LIN {X 0,Y 116.335,Z 316.276,A -85,B 0,C 180,E1 -30784.417,E2 -30784.417} C_VEL
LIN {X 0,Y 111.111,Z 327.603,A -85,B 0,C 180,E1 -30784.983,E2 -30784.983} C_VEL
LIN {X 0,Y 104.199,Z 339.212,A -85,B 0,C 180,E1 -30785.813,E2 -30785.813} C_VEL
LIN {X 0,Y 96.428,Z 349.65,A -85,B 0,C 180,E1 -30786.768,E2 -30786.768} C_VEL
LIN {X 0,Y 88.698,Z 358.177,A -85,B 0,C 180,E1 -30787.928,E2 -30787.928} C_VEL
LIN {X 0,Y 80.178,Z 366.031,A -85,B 0,C 180,E1 -30789.557,E2 -30789.557} C_VEL
LIN {X 0,Y 70.072,Z 373.698,A -85,B 0,C 180,E1 -30792.071,E2 -30792.071} C_VEL
LIN {X 0,Y 59.136,Z 380.359,A -85,B 0,C 180,E1 -30795.515,E2 -30795.515} C_VEL
LIN {X 0,Y 48.678,Z 385.44,A -85,B 0,C 180,E1 -30800.205,E2 -30800.205} C_VEL
LIN {X 0,Y 39.402,Z 389.024,A -85,B 0,C 180,E1 -30806.896,E2 -30806.896} C_VEL
LIN {X 0,Y 33.772,Z 390.828,A -85,B 0,C 180,E1 -30813.134,E2 -30813.134} C_VEL
LIN {X 0,Y 29.038,Z 392.153,A -85,B 0,C 180,E1 -30819.112,E2 -30819.112} C_VEL
LIN {X 0,Y 24.036,Z 393.133,A -85,B 0,C 180,E1 -30825.728,E2 -30825.728} C_VEL
LIN {X 0,Y 15.053,Z 394.132,A -85,B 0,C 180,E1 -30849.577,E2 -30849.577} C_VEL
LIN {X 0,Y 13.114,Z 394.223,A -85,B 0,C 180,E1 -30872.794,E2 -30872.794} C_VEL
LIN {X 0,Y 13.234,Z 394.154,A -85,B 0,C 180,E1 -30881.451,E2 -30881.451} C_VEL
LIN {X 0,Y 18.75,Z 393.445,A -85,B 0,C 180,E1 -30918.559,E2 -30918.559} C_VEL
LIN {X 0,Y 30.297,Z 391.115,A -85,B 0,C 180,E1 -30938.102,E2 -30938.102} C_VEL
LIN {X 0,Y 40.004,Z 388.239,A -85,B 0,C 180,E1 -30945.07,E2 -30945.07} C_VEL
LIN {X 0,Y 50.072,Z 384.335,A -85,B 0,C 180,E1 -30949.262,E2 -30949.262} C_VEL
LIN {X 0,Y 60.319,Z 379.297,A -85,B 0,C 180,E1 -30952.041,E2 -30952.041} C_VEL
LIN {X 0,Y 71.415,Z 372.402,A -85,B 0,C 180,E1 -30954.352,E2 -30954.352} C_VEL
LIN {X 0,Y 81.033,Z 365.019,A -85,B 0,C 180,E1 -30955.862,E2 -30955.862} C_VEL
LIN {X 0,Y 89.74,Z 356.925,A -85,B 0,C 180,E1 -30956.867,E2 -30956.867} C_VEL
LIN {X 0,Y 98.466,Z 347.049,A -85,B 0,C 180,E1 -30957.761,E2 -30957.761} C_VEL
LIN {X 0,Y 106.34,Z 335.913,A -85,B 0,C 180,E1 -30958.385,E2 -30958.385} C_VEL
LIN {X 0,Y 113.153,Z 323.625,A -85,B 0,C 180,E1 -30958.871,E2 -30958.871} C_VEL
LIN {X 0,Y 118.047,Z 312.096,A -85,B 0,C 180,E1 -30959.327,E2 -30959.327} C_VEL
LIN {X 0,Y 118.64,Z 310.381,A -85,B 0,C 180,E1 -30959.372,E2 -30959.372} C_VEL
LIN {X 0,Y 118.928,Z 309.527,A -85,B 0,C 180,E1 -30959.577,E2 -30959.577} C_VEL
LIN {X 0,Y 118.962,Z 309.436,A -85,B 0,C 180,E1 -30960,E2 -30960} C_VEL
LIN {X 0,Y 118.673,Z 310.311,A -85,B 0,C 180,E1 -30960.312,E2 -30960.312} C_VEL
LIN {X 0,Y 113.846,Z 322.247,A -85,B 0,C 180,E1 -30960.541,E2 -30960.541} C_VEL
LIN {X 0,Y 107.19,Z 334.592,A -85,B 0,C 180,E1 -30960.931,E2 -30960.931} C_VEL
LIN {X 0,Y 99.301,Z 346.079,A -85,B 0,C 180,E1 -30961.448,E2 -30961.448} C_VEL
LIN {X 0,Y 91.419,Z 355.322,A -85,B 0,C 180,E1 -30962.004,E2 -30962.004} C_VEL
LIN {X 0,Y 82.68,Z 363.758,A -85,B 0,C 180,E1 -30962.848,E2 -30962.848} C_VEL
LIN {X 0,Y 72.227,Z 372.001,A -85,B 0,C 180,E1 -30964.163,E2 -30964.163} C_VEL
LIN {X 0,Y 61.835,Z 378.65,A -85,B 0,C 180,E1 -30966.032,E2 -30966.032} C_VEL
LIN {X 0,Y 49.848,Z 384.729,A -85,B 0,C 180,E1 -30969.281,E2 -30969.281} C_VEL
LIN {X 0,Y 39.719,Z 388.681,A -85,B 0,C 180,E1 -30973.303,E2 -30973.303} C_VEL
LIN {X 0,Y 29.9,Z 391.604,A -85,B 0,C 180,E1 -30979.915,E2 -30979.915} C_VEL
LIN {X 0,Y 18.311,Z 393.995,A -85,B 0,C 180,E1 -30999.86,E2 -30999.86} C_VEL
LIN {X 0,Y 14.211,Z 394.606,A -85,B 0,C 180,E1 -31020.362,E2 -31020.362} C_VEL
LIN {X 0,Y 12.854,Z 394.82,A -85,B 0,C 180,E1 -31050.001,E2 -31050.001} C_VEL
LIN {X 0,Y 14.252,Z 394.584,A -85,B 0,C 180,E1 -31079.548,E2 -31079.548} C_VEL
LIN {X 0,Y 23.782,Z 392.946,A -85,B 0,C 180,E1 -31112.443,E2 -31112.443} C_VEL
LIN {X 0,Y 29.9,Z 391.53,A -85,B 0,C 180,E1 -31120.086,E2 -31120.086} C_VEL
LIN {X 0,Y 39.72,Z 388.577,A -85,B 0,C 180,E1 -31126.699,E2 -31126.699} C_VEL
LIN {X 0,Y 49.846,Z 384.587,A -85,B 0,C 180,E1 -31130.737,E2 -31130.737} C_VEL
LIN {X 0,Y 61.66,Z 378.551,A -85,B 0,C 180,E1 -31133.979,E2 -31133.979} C_VEL
LIN {X 0,Y 72.227,Z 371.759,A -85,B 0,C 180,E1 -31135.848,E2 -31135.848} C_VEL
LIN {X 0,Y 82.68,Z 363.464,A -85,B 0,C 180,E1 -31137.166,E2 -31137.166} C_VEL
LIN {X 0,Y 91.418,Z 354.949,A -85,B 0,C 180,E1 -31138.022,E2 -31138.022} C_VEL
LIN {X 0,Y 100.176,Z 344.435,A -85,B 0,C 180,E1 -31138.663,E2 -31138.663} C_VEL
LIN {X 0,Y 107.19,Z 334.027,A -85,B 0,C 180,E1 -31139.095,E2 -31139.095} C_VEL
LIN {X 0,Y 113.494,Z 322.249,A -85,B 0,C 180,E1 -31139.458,E2 -31139.458} C_VEL
LIN {X 0,Y 118.382,Z 310.126,A -85,B 0,C 180,E1 -31139.661,E2 -31139.661} C_VEL
LIN {X 0,Y 118.695,Z 309.179,A -85,B 0,C 180,E1 -31140,E2 -31140} C_VEL
LIN {X 0,Y 118.688,Z 309.187,A -85,B 0,C 180,E1 -31140.424,E2 -31140.424} C_VEL
LIN {X 0,Y 118.123,Z 310.864,A -85,B 0,C 180,E1 -31140.71,E2 -31140.71} C_VEL
LIN {X 0,Y 113.082,Z 323.059,A -85,B 0,C 180,E1 -31141.171,E2 -31141.171} C_VEL
LIN {X 0,Y 107.22,Z 333.916,A -85,B 0,C 180,E1 -31141.623,E2 -31141.623} C_VEL
LIN {X 0,Y 99.346,Z 345.463,A -85,B 0,C 180,E1 -31142.234,E2 -31142.234} C_VEL
LIN {X 0,Y 91.489,Z 354.765,A -85,B 0,C 180,E1 -31142.996,E2 -31142.996} C_VEL
LIN {X 0,Y 82.779,Z 363.236,A -85,B 0,C 180,E1 -31143.985,E2 -31143.985} C_VEL
LIN {X 0,Y 72.726,Z 371.231,A -85,B 0,C 180,E1 -31145.546,E2 -31145.546} C_VEL
LIN {X 0,Y 63.759,Z 377.109,A -85,B 0,C 180,E1 -31147.228,E2 -31147.228} C_VEL
LIN {X 0,Y 53.488,Z 382.601,A -85,B 0,C 180,E1 -31149.782,E2 -31149.782} C_VEL
LIN {X 0,Y 43.334,Z 386.911,A -85,B 0,C 180,E1 -31153.323,E2 -31153.323} C_VEL
LIN {X 0,Y 36.732,Z 389.188,A -85,B 0,C 180,E1 -31156.931,E2 -31156.931} C_VEL
LIN {X 0,Y 29.98,Z 391.11,A -85,B 0,C 180,E1 -31162.328,E2 -31162.328} C_VEL
LIN {X 0,Y 24.239,Z 392.42,A -85,B 0,C 180,E1 -31169.558,E2 -31169.558} C_VEL
LIN {X 0,Y 14.632,Z 394.007,A -85,B 0,C 180,E1 -31201.293,E2 -31201.293} C_VEL
LIN {X 0,Y 13.234,Z 394.154,A -85,B 0,C 180,E1 -31241.451,E2 -31241.451} C_VEL
LIN {X 0,Y 14.731,Z 393.966,A -85,B 0,C 180,E1 -31265.019,E2 -31265.019} C_VEL
LIN {X 0,Y 19.691,Z 393.091,A -85,B 0,C 180,E1 -31294.072,E2 -31294.072} C_VEL
LIN {X 0,Y 25.62,Z 391.889,A -85,B 0,C 180,E1 -31307.406,E2 -31307.406} C_VEL
LIN {X 0,Y 30.873,Z 390.659,A -85,B 0,C 180,E1 -31312.487,E2 -31312.487} C_VEL
LIN {X 0,Y 32.732,Z 390.137,A -85,B 0,C 180,E1 -31313.378,E2 -31313.378} C_VEL
LIN {X 0,Y 42.263,Z 387.2,A -85,B 0,C 180,E1 -31316.149,E2 -31316.149} C_VEL
LIN {X 0,Y 52.745,Z 382.929,A -85,B 0,C 180,E1 -31317.903,E2 -31317.903} C_VEL
LIN {X 0,Y 56.246,Z 381.26,A -85,B 0,C 180,E1 -31318.384,E2 -31318.384} C_VEL
LIN {X 0,Y 56.579,Z 381.113,A -85,B 0,C 180,E1 -31320,E2 -31320} C_VEL
LIN {X 0,Y 45.699,Z 385.999,A -85,B 0,C 180,E1 -31321.565,E2 -31321.565} C_VEL
LIN {X 0,Y 35.22,Z 389.591,A -85,B 0,C 180,E1 -31323.869,E2 -31323.869} C_VEL
LIN {X 0,Y 28.278,Z 391.442,A -85,B 0,C 180,E1 -31326.213,E2 -31326.213} C_VEL
LIN {X 0,Y 14.792,Z 393.833,A -85,B 0,C 180,E1 -31338.161,E2 -31338.161} C_VEL
LIN {X 0,Y 8.773,Z 394.444,A -85,B 0,C 180,E1 -31356.769,E2 -31356.769} C_VEL
LIN {X 0,Y 5.742,Z 394.657,A -85,B 0,C 180,E1 -31410.003,E2 -31410.003} C_VEL
LIN {X 0,Y 8.796,Z 394.421,A -85,B 0,C 180,E1 -31463.04,E2 -31463.04} C_VEL
LIN {X 0,Y 21.434,Z 392.782,A -85,B 0,C 180,E1 -31489.637,E2 -31489.637} C_VEL
LIN {X 0,Y 28.278,Z 391.366,A -85,B 0,C 180,E1 -31493.788,E2 -31493.788} C_VEL
LIN {X 0,Y 38.707,Z 388.413,A -85,B 0,C 180,E1 -31497.017,E2 -31497.017} C_VEL
LIN {X 0,Y 51.701,Z 383.289,A -85,B 0,C 180,E1 -31499.346,E2 -31499.346} C_VEL
LIN {X 0,Y 56.224,Z 381.114,A -85,B 0,C 180,E1 -31500,E2 -31500} C_VEL
LIN {X 0,Y 56.249,Z 381.076,A -85,B 0,C 180,E1 -31501.7,E2 -31501.7} C_VEL
LIN {X 0,Y 45.757,Z 385.767,A -85,B 0,C 180,E1 -31503.272,E2 -31503.272} C_VEL
LIN {X 0,Y 35.321,Z 389.352,A -85,B 0,C 180,E1 -31505.803,E2 -31505.803} C_VEL
LIN {X 0,Y 28.431,Z 391.199,A -85,B 0,C 180,E1 -31508.588,E2 -31508.588} C_VEL
LIN {X 0,Y 21.632,Z 392.583,A -85,B 0,C 180,E1 -31512.927,E2 -31512.927} C_VEL
LIN {X 0,Y 9.068,Z 394.169,A -85,B 0,C 180,E1 -31539.191,E2 -31539.191} C_VEL
LIN {X 0,Y 6.351,Z 394.323,A -85,B 0,C 180,E1 -31612.18,E2 -31612.18} C_VEL
LIN {X 0,Y 15.025,Z 393.607,A -85,B 0,C 180,E1 -31659.308,E2 -31659.308} C_VEL
LIN {X 0,Y 28.423,Z 391.277,A -85,B 0,C 180,E1 -31671.516,E2 -31671.516} C_VEL
LIN {X 0,Y 32.732,Z 390.137,A -85,B 0,C 180,E1 -31673.378,E2 -31673.378} C_VEL
LIN {X 0,Y 35.18,Z 392.074,A -85,B 0,C 180,E1 -31674.228,E2 -31674.228} C_VEL
LIN {X 0,Y 35.18,Z 600,A -85,B 0,C 180,E1 -31674.228,E2 -31674.228} C_VEL
LIN {X 0,Y 35.18,Z 600,A -85,B 0,C 180,E1 -31674.228,E2 -31674.228}

QRS_NEXT_CUT()

QRS_NEXT()
QRS_HOME()

END
